// TIA Portal V18 export
// export: Created 2026-06-20T13:30:08.8484285Z, ExportSetting WithDefaults, DisplayName Totally Integrated Automation Portal, DisplayVersion V18, DisplayName TIA Portal Openness, DisplayVersion V18, DisplayName TIA Portal Version Control Interface, DisplayVersion V18, DisplayName STEP 7 Professional, DisplayVersion V18, DisplayName STEP 7 Safety, DisplayVersion V18, DisplayName WinCC Professional, DisplayVersion V18
FUNCTION "FC_HMI_Mirror_PLC1" : Void   // FC40, LAD
{ S7_Optimized_Access := 'TRUE' }
VERSION : 0.1
// stored: AutoNumber true, IsIECCheckEnabled false, SetENOAutomatically false, UDAEnableTagReadback false
BEGIN

REGION Network 1: Mirror V3230_Nuoc_Bon1
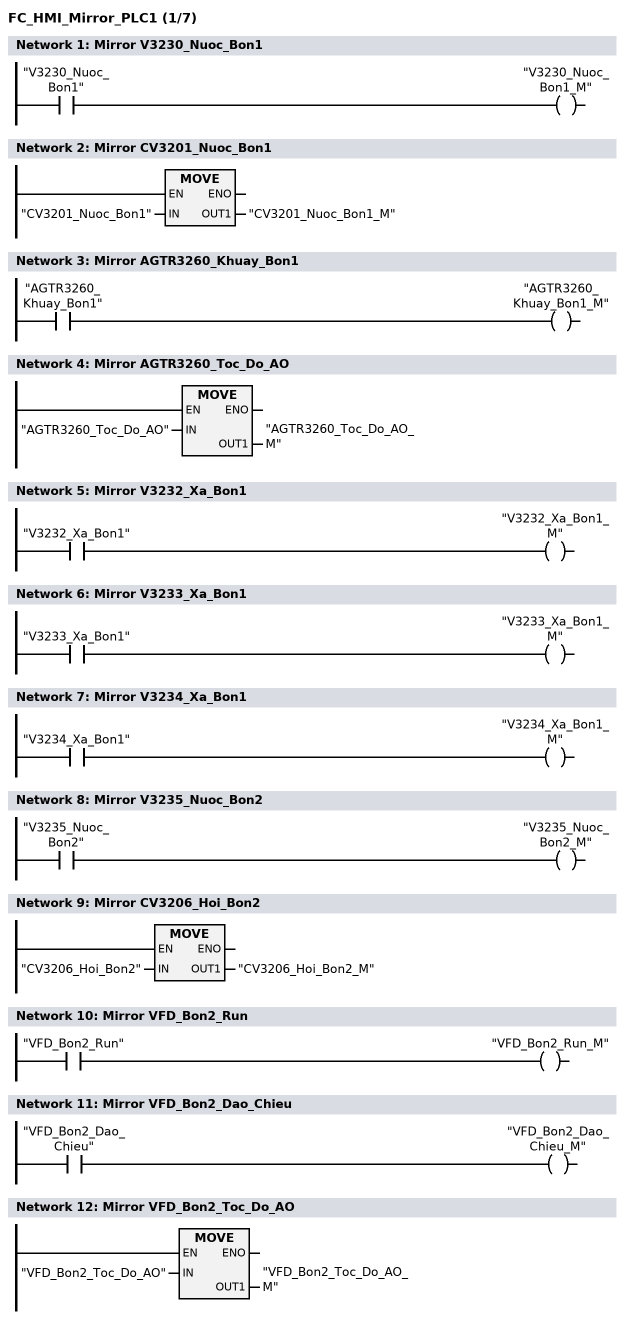
   RUNG wire#powerrail
      Contact( "V3230_Nuoc_Bon1" )
      Coil( "V3230_Nuoc_Bon1_M" )
   END_RUNG
   // the same network as SCL:
   "V3230_Nuoc_Bon1_M" := "V3230_Nuoc_Bon1";
END_REGION

REGION Network 2: Mirror CV3201_Nuoc_Bon1
   RUNG wire#powerrail
      { S7_GenerateENO := "TRUE" } Move(in := "CV3201_Nuoc_Bon1", out1 => "CV3201_Nuoc_Bon1_M")
   END_RUNG
   // the same network as SCL:
   "CV3201_Nuoc_Bon1_M" := "CV3201_Nuoc_Bon1";
END_REGION

REGION Network 3: Mirror AGTR3260_Khuay_Bon1
   RUNG wire#powerrail
      Contact( "AGTR3260_Khuay_Bon1" )
      Coil( "AGTR3260_Khuay_Bon1_M" )
   END_RUNG
   // the same network as SCL:
   "AGTR3260_Khuay_Bon1_M" := "AGTR3260_Khuay_Bon1";
END_REGION

REGION Network 4: Mirror AGTR3260_Toc_Do_AO
   RUNG wire#powerrail
      { S7_GenerateENO := "TRUE" } Move(in := "AGTR3260_Toc_Do_AO", out1 => "AGTR3260_Toc_Do_AO_M")
   END_RUNG
   // the same network as SCL:
   "AGTR3260_Toc_Do_AO_M" := "AGTR3260_Toc_Do_AO";
END_REGION

REGION Network 5: Mirror V3232_Xa_Bon1
   RUNG wire#powerrail
      Contact( "V3232_Xa_Bon1" )
      Coil( "V3232_Xa_Bon1_M" )
   END_RUNG
   // the same network as SCL:
   "V3232_Xa_Bon1_M" := "V3232_Xa_Bon1";
END_REGION

REGION Network 6: Mirror V3233_Xa_Bon1
   RUNG wire#powerrail
      Contact( "V3233_Xa_Bon1" )
      Coil( "V3233_Xa_Bon1_M" )
   END_RUNG
   // the same network as SCL:
   "V3233_Xa_Bon1_M" := "V3233_Xa_Bon1";
END_REGION

REGION Network 7: Mirror V3234_Xa_Bon1
   RUNG wire#powerrail
      Contact( "V3234_Xa_Bon1" )
      Coil( "V3234_Xa_Bon1_M" )
   END_RUNG
   // the same network as SCL:
   "V3234_Xa_Bon1_M" := "V3234_Xa_Bon1";
END_REGION

REGION Network 8: Mirror V3235_Nuoc_Bon2
   RUNG wire#powerrail
      Contact( "V3235_Nuoc_Bon2" )
      Coil( "V3235_Nuoc_Bon2_M" )
   END_RUNG
   // the same network as SCL:
   "V3235_Nuoc_Bon2_M" := "V3235_Nuoc_Bon2";
END_REGION

REGION Network 9: Mirror CV3206_Hoi_Bon2
   RUNG wire#powerrail
      { S7_GenerateENO := "TRUE" } Move(in := "CV3206_Hoi_Bon2", out1 => "CV3206_Hoi_Bon2_M")
   END_RUNG
   // the same network as SCL:
   "CV3206_Hoi_Bon2_M" := "CV3206_Hoi_Bon2";
END_REGION

REGION Network 10: Mirror VFD_Bon2_Run
   RUNG wire#powerrail
      Contact( "VFD_Bon2_Run" )
      Coil( "VFD_Bon2_Run_M" )
   END_RUNG
   // the same network as SCL:
   "VFD_Bon2_Run_M" := "VFD_Bon2_Run";
END_REGION

REGION Network 11: Mirror VFD_Bon2_Dao_Chieu
   RUNG wire#powerrail
      Contact( "VFD_Bon2_Dao_Chieu" )
      Coil( "VFD_Bon2_Dao_Chieu_M" )
   END_RUNG
   // the same network as SCL:
   "VFD_Bon2_Dao_Chieu_M" := "VFD_Bon2_Dao_Chieu";
END_REGION

REGION Network 12: Mirror VFD_Bon2_Toc_Do_AO
   RUNG wire#powerrail
      { S7_GenerateENO := "TRUE" } Move(in := "VFD_Bon2_Toc_Do_AO", out1 => "VFD_Bon2_Toc_Do_AO_M")
   END_RUNG
   // the same network as SCL:
   "VFD_Bon2_Toc_Do_AO_M" := "VFD_Bon2_Toc_Do_AO";
END_REGION

REGION Network 13: Mirror V3237_Xa_Bon2
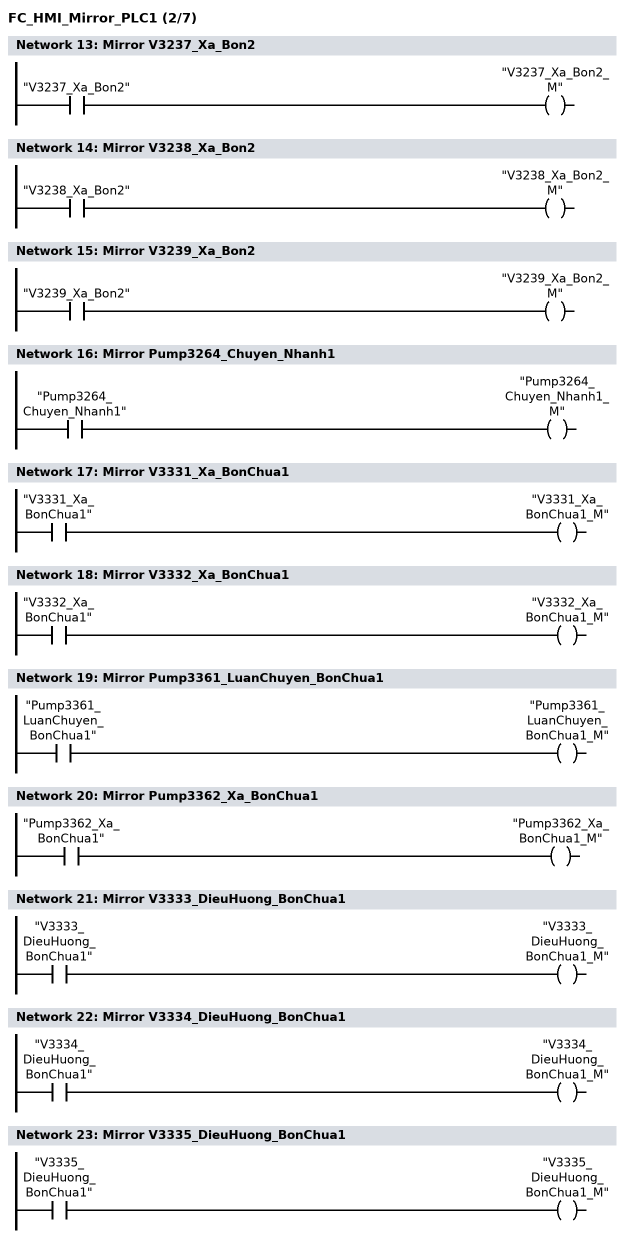
   RUNG wire#powerrail
      Contact( "V3237_Xa_Bon2" )
      Coil( "V3237_Xa_Bon2_M" )
   END_RUNG
   // the same network as SCL:
   "V3237_Xa_Bon2_M" := "V3237_Xa_Bon2";
END_REGION

REGION Network 14: Mirror V3238_Xa_Bon2
   RUNG wire#powerrail
      Contact( "V3238_Xa_Bon2" )
      Coil( "V3238_Xa_Bon2_M" )
   END_RUNG
   // the same network as SCL:
   "V3238_Xa_Bon2_M" := "V3238_Xa_Bon2";
END_REGION

REGION Network 15: Mirror V3239_Xa_Bon2
   RUNG wire#powerrail
      Contact( "V3239_Xa_Bon2" )
      Coil( "V3239_Xa_Bon2_M" )
   END_RUNG
   // the same network as SCL:
   "V3239_Xa_Bon2_M" := "V3239_Xa_Bon2";
END_REGION

REGION Network 16: Mirror Pump3264_Chuyen_Nhanh1
   RUNG wire#powerrail
      Contact( "Pump3264_Chuyen_Nhanh1" )
      Coil( "Pump3264_Chuyen_Nhanh1_M" )
   END_RUNG
   // the same network as SCL:
   "Pump3264_Chuyen_Nhanh1_M" := "Pump3264_Chuyen_Nhanh1";
END_REGION

REGION Network 17: Mirror V3331_Xa_BonChua1
   RUNG wire#powerrail
      Contact( "V3331_Xa_BonChua1" )
      Coil( "V3331_Xa_BonChua1_M" )
   END_RUNG
   // the same network as SCL:
   "V3331_Xa_BonChua1_M" := "V3331_Xa_BonChua1";
END_REGION

REGION Network 18: Mirror V3332_Xa_BonChua1
   RUNG wire#powerrail
      Contact( "V3332_Xa_BonChua1" )
      Coil( "V3332_Xa_BonChua1_M" )
   END_RUNG
   // the same network as SCL:
   "V3332_Xa_BonChua1_M" := "V3332_Xa_BonChua1";
END_REGION

REGION Network 19: Mirror Pump3361_LuanChuyen_BonChua1
   RUNG wire#powerrail
      Contact( "Pump3361_LuanChuyen_BonChua1" )
      Coil( "Pump3361_LuanChuyen_BonChua1_M" )
   END_RUNG
   // the same network as SCL:
   "Pump3361_LuanChuyen_BonChua1_M" := "Pump3361_LuanChuyen_BonChua1";
END_REGION

REGION Network 20: Mirror Pump3362_Xa_BonChua1
   RUNG wire#powerrail
      Contact( "Pump3362_Xa_BonChua1" )
      Coil( "Pump3362_Xa_BonChua1_M" )
   END_RUNG
   // the same network as SCL:
   "Pump3362_Xa_BonChua1_M" := "Pump3362_Xa_BonChua1";
END_REGION

REGION Network 21: Mirror V3333_DieuHuong_BonChua1
   RUNG wire#powerrail
      Contact( "V3333_DieuHuong_BonChua1" )
      Coil( "V3333_DieuHuong_BonChua1_M" )
   END_RUNG
   // the same network as SCL:
   "V3333_DieuHuong_BonChua1_M" := "V3333_DieuHuong_BonChua1";
END_REGION

REGION Network 22: Mirror V3334_DieuHuong_BonChua1
   RUNG wire#powerrail
      Contact( "V3334_DieuHuong_BonChua1" )
      Coil( "V3334_DieuHuong_BonChua1_M" )
   END_RUNG
   // the same network as SCL:
   "V3334_DieuHuong_BonChua1_M" := "V3334_DieuHuong_BonChua1";
END_REGION

REGION Network 23: Mirror V3335_DieuHuong_BonChua1
   RUNG wire#powerrail
      Contact( "V3335_DieuHuong_BonChua1" )
      Coil( "V3335_DieuHuong_BonChua1_M" )
   END_RUNG
   // the same network as SCL:
   "V3335_DieuHuong_BonChua1_M" := "V3335_DieuHuong_BonChua1";
END_REGION

REGION Network 24: Mirror CV3304_Nuoc_Lam_Mat
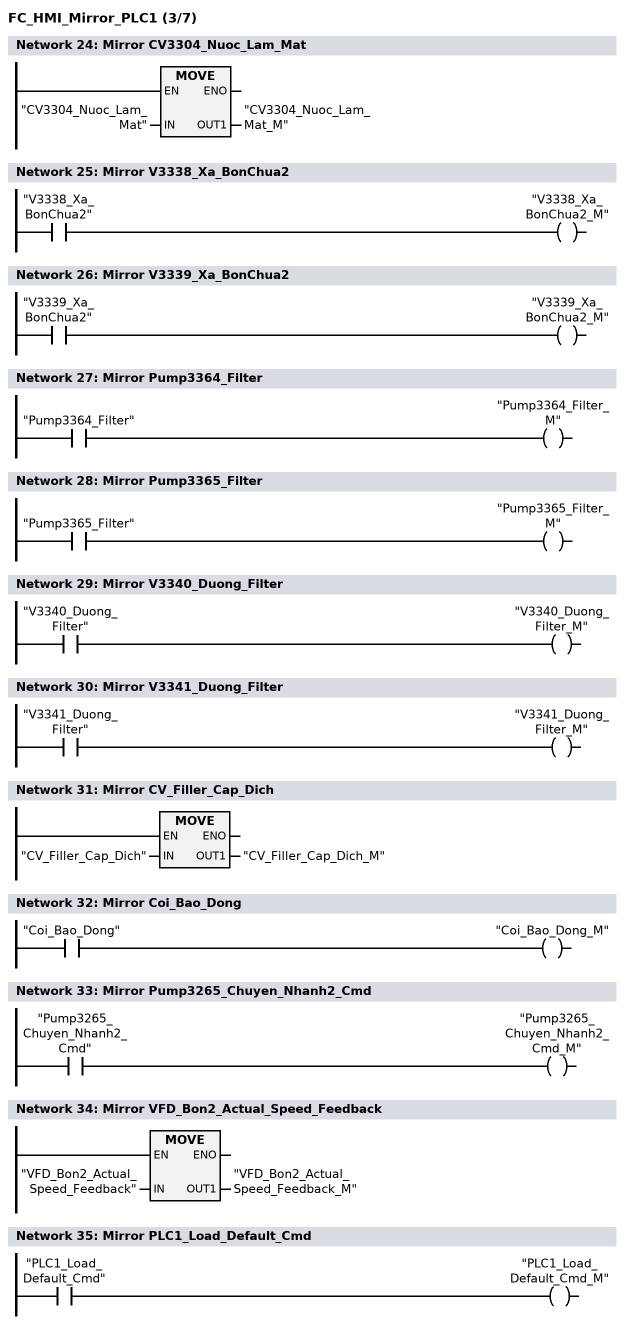
   RUNG wire#powerrail
      { S7_GenerateENO := "TRUE" } Move(in := "CV3304_Nuoc_Lam_Mat", out1 => "CV3304_Nuoc_Lam_Mat_M")
   END_RUNG
   // the same network as SCL:
   "CV3304_Nuoc_Lam_Mat_M" := "CV3304_Nuoc_Lam_Mat";
END_REGION

REGION Network 25: Mirror V3338_Xa_BonChua2
   RUNG wire#powerrail
      Contact( "V3338_Xa_BonChua2" )
      Coil( "V3338_Xa_BonChua2_M" )
   END_RUNG
   // the same network as SCL:
   "V3338_Xa_BonChua2_M" := "V3338_Xa_BonChua2";
END_REGION

REGION Network 26: Mirror V3339_Xa_BonChua2
   RUNG wire#powerrail
      Contact( "V3339_Xa_BonChua2" )
      Coil( "V3339_Xa_BonChua2_M" )
   END_RUNG
   // the same network as SCL:
   "V3339_Xa_BonChua2_M" := "V3339_Xa_BonChua2";
END_REGION

REGION Network 27: Mirror Pump3364_Filter
   RUNG wire#powerrail
      Contact( "Pump3364_Filter" )
      Coil( "Pump3364_Filter_M" )
   END_RUNG
   // the same network as SCL:
   "Pump3364_Filter_M" := "Pump3364_Filter";
END_REGION

REGION Network 28: Mirror Pump3365_Filter
   RUNG wire#powerrail
      Contact( "Pump3365_Filter" )
      Coil( "Pump3365_Filter_M" )
   END_RUNG
   // the same network as SCL:
   "Pump3365_Filter_M" := "Pump3365_Filter";
END_REGION

REGION Network 29: Mirror V3340_Duong_Filter
   RUNG wire#powerrail
      Contact( "V3340_Duong_Filter" )
      Coil( "V3340_Duong_Filter_M" )
   END_RUNG
   // the same network as SCL:
   "V3340_Duong_Filter_M" := "V3340_Duong_Filter";
END_REGION

REGION Network 30: Mirror V3341_Duong_Filter
   RUNG wire#powerrail
      Contact( "V3341_Duong_Filter" )
      Coil( "V3341_Duong_Filter_M" )
   END_RUNG
   // the same network as SCL:
   "V3341_Duong_Filter_M" := "V3341_Duong_Filter";
END_REGION

REGION Network 31: Mirror CV_Filler_Cap_Dich
   RUNG wire#powerrail
      { S7_GenerateENO := "TRUE" } Move(in := "CV_Filler_Cap_Dich", out1 => "CV_Filler_Cap_Dich_M")
   END_RUNG
   // the same network as SCL:
   "CV_Filler_Cap_Dich_M" := "CV_Filler_Cap_Dich";
END_REGION

REGION Network 32: Mirror Coi_Bao_Dong
   RUNG wire#powerrail
      Contact( "Coi_Bao_Dong" )
      Coil( "Coi_Bao_Dong_M" )
   END_RUNG
   // the same network as SCL:
   "Coi_Bao_Dong_M" := "Coi_Bao_Dong";
END_REGION

REGION Network 33: Mirror Pump3265_Chuyen_Nhanh2_Cmd
   RUNG wire#powerrail
      Contact( "Pump3265_Chuyen_Nhanh2_Cmd" )
      Coil( "Pump3265_Chuyen_Nhanh2_Cmd_M" )
   END_RUNG
   // the same network as SCL:
   "Pump3265_Chuyen_Nhanh2_Cmd_M" := "Pump3265_Chuyen_Nhanh2_Cmd";
END_REGION

REGION Network 34: Mirror VFD_Bon2_Actual_Speed_Feedback
   RUNG wire#powerrail
      { S7_GenerateENO := "TRUE" } Move(in := "VFD_Bon2_Actual_Speed_Feedback", out1 => "VFD_Bon2_Actual_Speed_Feedback_M")
   END_RUNG
   // the same network as SCL:
   "VFD_Bon2_Actual_Speed_Feedback_M" := "VFD_Bon2_Actual_Speed_Feedback";
END_REGION

REGION Network 35: Mirror PLC1_Load_Default_Cmd
   RUNG wire#powerrail
      Contact( "PLC1_Load_Default_Cmd" )
      Coil( "PLC1_Load_Default_Cmd_M" )
   END_RUNG
   // the same network as SCL:
   "PLC1_Load_Default_Cmd_M" := "PLC1_Load_Default_Cmd";
END_REGION

REGION Network 36: Quyền Operator
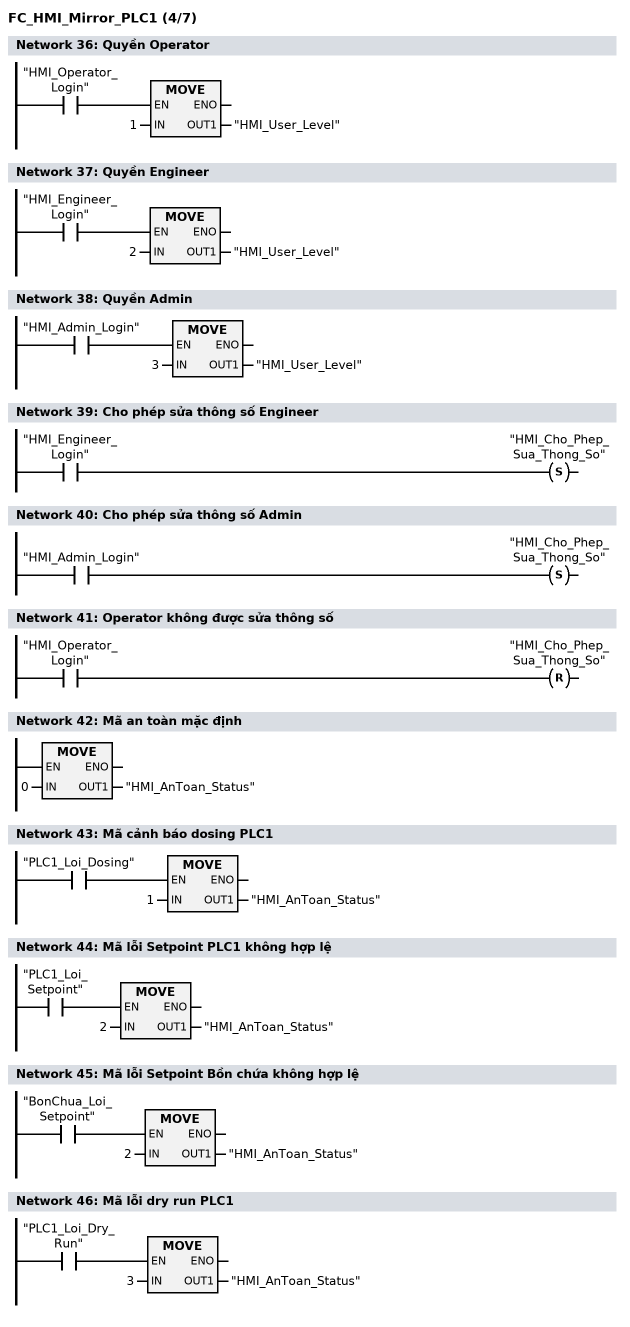
   RUNG wire#powerrail
      Contact( "HMI_Operator_Login" )
      { S7_GenerateENO := "TRUE" } Move(in := 1, out1 => "HMI_User_Level")
   END_RUNG
   // the same network as SCL:
   IF "HMI_Operator_Login" THEN "HMI_User_Level" := 1; END_IF;
END_REGION

REGION Network 37: Quyền Engineer
   RUNG wire#powerrail
      Contact( "HMI_Engineer_Login" )
      { S7_GenerateENO := "TRUE" } Move(in := 2, out1 => "HMI_User_Level")
   END_RUNG
   // the same network as SCL:
   IF "HMI_Engineer_Login" THEN "HMI_User_Level" := 2; END_IF;
END_REGION

REGION Network 38: Quyền Admin
   RUNG wire#powerrail
      Contact( "HMI_Admin_Login" )
      { S7_GenerateENO := "TRUE" } Move(in := 3, out1 => "HMI_User_Level")
   END_RUNG
   // the same network as SCL:
   IF "HMI_Admin_Login" THEN "HMI_User_Level" := 3; END_IF;
END_REGION

REGION Network 39: Cho phép sửa thông số Engineer
   RUNG wire#powerrail
      Contact( "HMI_Engineer_Login" )
      S_Coil( "HMI_Cho_Phep_Sua_Thong_So" )
   END_RUNG
   // the same network as SCL:
   IF "HMI_Engineer_Login" THEN "HMI_Cho_Phep_Sua_Thong_So" := TRUE; END_IF;
END_REGION

REGION Network 40: Cho phép sửa thông số Admin
   RUNG wire#powerrail
      Contact( "HMI_Admin_Login" )
      S_Coil( "HMI_Cho_Phep_Sua_Thong_So" )
   END_RUNG
   // the same network as SCL:
   IF "HMI_Admin_Login" THEN "HMI_Cho_Phep_Sua_Thong_So" := TRUE; END_IF;
END_REGION

REGION Network 41: Operator không được sửa thông số
   RUNG wire#powerrail
      Contact( "HMI_Operator_Login" )
      R_Coil( "HMI_Cho_Phep_Sua_Thong_So" )
   END_RUNG
   // the same network as SCL:
   IF "HMI_Operator_Login" THEN "HMI_Cho_Phep_Sua_Thong_So" := FALSE; END_IF;
END_REGION

REGION Network 42: Mã an toàn mặc định
   RUNG wire#powerrail
      { S7_GenerateENO := "TRUE" } Move(in := 0, out1 => "HMI_AnToan_Status")
   END_RUNG
   // the same network as SCL:
   "HMI_AnToan_Status" := 0;
END_REGION

REGION Network 43: Mã cảnh báo dosing PLC1
   RUNG wire#powerrail
      Contact( "PLC1_Loi_Dosing" )
      { S7_GenerateENO := "TRUE" } Move(in := 1, out1 => "HMI_AnToan_Status")
   END_RUNG
   // the same network as SCL:
   IF "PLC1_Loi_Dosing" THEN "HMI_AnToan_Status" := 1; END_IF;
END_REGION

REGION Network 44: Mã lỗi Setpoint PLC1 không hợp lệ
   RUNG wire#powerrail
      Contact( "PLC1_Loi_Setpoint" )
      { S7_GenerateENO := "TRUE" } Move(in := 2, out1 => "HMI_AnToan_Status")
   END_RUNG
   // the same network as SCL:
   IF "PLC1_Loi_Setpoint" THEN "HMI_AnToan_Status" := 2; END_IF;
END_REGION

REGION Network 45: Mã lỗi Setpoint Bồn chứa không hợp lệ
   RUNG wire#powerrail
      Contact( "BonChua_Loi_Setpoint" )
      { S7_GenerateENO := "TRUE" } Move(in := 2, out1 => "HMI_AnToan_Status")
   END_RUNG
   // the same network as SCL:
   IF "BonChua_Loi_Setpoint" THEN "HMI_AnToan_Status" := 2; END_IF;
END_REGION

REGION Network 46: Mã lỗi dry run PLC1
   RUNG wire#powerrail
      Contact( "PLC1_Loi_Dry_Run" )
      { S7_GenerateENO := "TRUE" } Move(in := 3, out1 => "HMI_AnToan_Status")
   END_RUNG
   // the same network as SCL:
   IF "PLC1_Loi_Dry_Run" THEN "HMI_AnToan_Status" := 3; END_IF;
END_REGION

REGION Network 47: Mã E-Stop ưu tiên cao PLC1
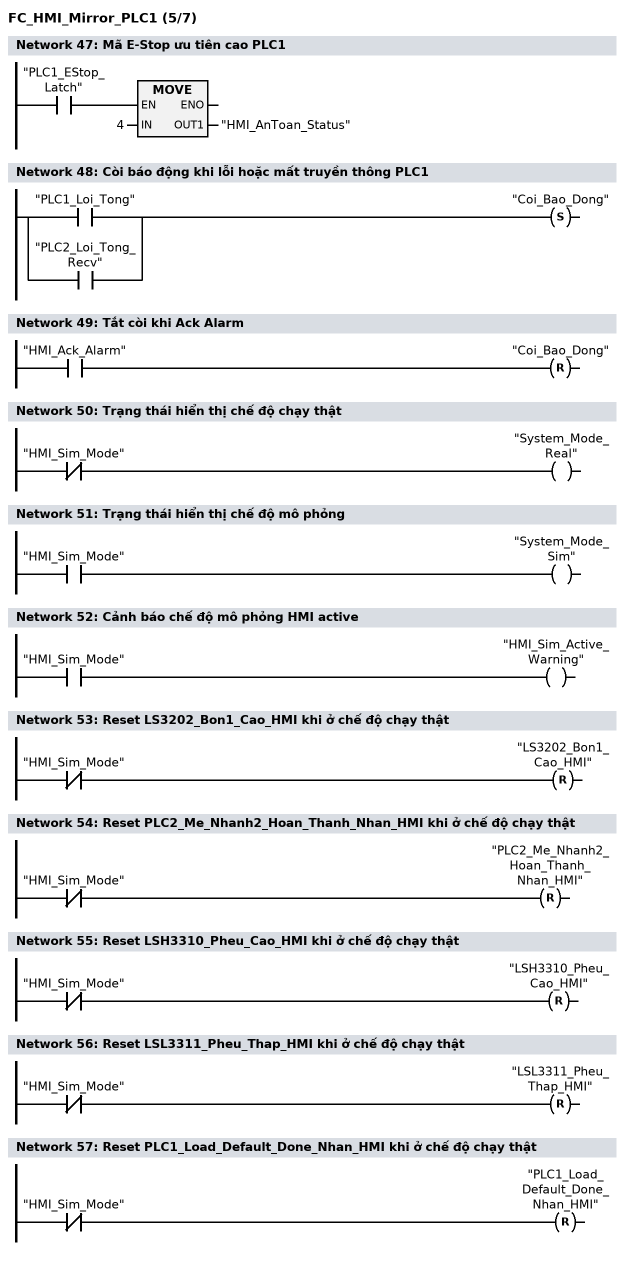
   RUNG wire#powerrail
      Contact( "PLC1_EStop_Latch" )
      { S7_GenerateENO := "TRUE" } Move(in := 4, out1 => "HMI_AnToan_Status")
   END_RUNG
   // the same network as SCL:
   IF "PLC1_EStop_Latch" THEN "HMI_AnToan_Status" := 4; END_IF;
END_REGION

REGION Network 48: Còi báo động khi lỗi hoặc mất truyền thông PLC1
   RUNG wire#powerrail
      Contact( "PLC1_Loi_Tong" )
      wire#w1
      S_Coil( "Coi_Bao_Dong" )
   END_RUNG
   RUNG wire#powerrail
      Contact( "PLC2_Loi_Tong_Recv" )
   END_RUNG wire#w1
   // the same network as SCL:
   IF "PLC1_Loi_Tong" OR "PLC2_Loi_Tong_Recv" THEN "Coi_Bao_Dong" := TRUE; END_IF;
END_REGION

REGION Network 49: Tắt còi khi Ack Alarm
   RUNG wire#powerrail
      Contact( "HMI_Ack_Alarm" )
      R_Coil( "Coi_Bao_Dong" )
   END_RUNG
   // the same network as SCL:
   IF "HMI_Ack_Alarm" THEN "Coi_Bao_Dong" := FALSE; END_IF;
END_REGION

REGION Network 50: Trạng thái hiển thị chế độ chạy thật
   RUNG wire#powerrail
      I_Contact( "HMI_Sim_Mode" )
      Coil( "System_Mode_Real" )
   END_RUNG
   // the same network as SCL:
   "System_Mode_Real" := NOT "HMI_Sim_Mode";
END_REGION

REGION Network 51: Trạng thái hiển thị chế độ mô phỏng
   RUNG wire#powerrail
      Contact( "HMI_Sim_Mode" )
      Coil( "System_Mode_Sim" )
   END_RUNG
   // the same network as SCL:
   "System_Mode_Sim" := "HMI_Sim_Mode";
END_REGION

REGION Network 52: Cảnh báo chế độ mô phỏng HMI active
   RUNG wire#powerrail
      Contact( "HMI_Sim_Mode" )
      Coil( "HMI_Sim_Active_Warning" )
   END_RUNG
   // the same network as SCL:
   "HMI_Sim_Active_Warning" := "HMI_Sim_Mode";
END_REGION

REGION Network 53: Reset LS3202_Bon1_Cao_HMI khi ở chế độ chạy thật
   RUNG wire#powerrail
      I_Contact( "HMI_Sim_Mode" )
      R_Coil( "LS3202_Bon1_Cao_HMI" )
   END_RUNG
   // the same network as SCL:
   IF NOT "HMI_Sim_Mode" THEN "LS3202_Bon1_Cao_HMI" := FALSE; END_IF;
END_REGION

REGION Network 54: Reset PLC2_Me_Nhanh2_Hoan_Thanh_Nhan_HMI khi ở chế độ chạy thật
   RUNG wire#powerrail
      I_Contact( "HMI_Sim_Mode" )
      R_Coil( "PLC2_Me_Nhanh2_Hoan_Thanh_Nhan_HMI" )
   END_RUNG
   // the same network as SCL:
   IF NOT "HMI_Sim_Mode" THEN "PLC2_Me_Nhanh2_Hoan_Thanh_Nhan_HMI" := FALSE; END_IF;
END_REGION

REGION Network 55: Reset LSH3310_Pheu_Cao_HMI khi ở chế độ chạy thật
   RUNG wire#powerrail
      I_Contact( "HMI_Sim_Mode" )
      R_Coil( "LSH3310_Pheu_Cao_HMI" )
   END_RUNG
   // the same network as SCL:
   IF NOT "HMI_Sim_Mode" THEN "LSH3310_Pheu_Cao_HMI" := FALSE; END_IF;
END_REGION

REGION Network 56: Reset LSL3311_Pheu_Thap_HMI khi ở chế độ chạy thật
   RUNG wire#powerrail
      I_Contact( "HMI_Sim_Mode" )
      R_Coil( "LSL3311_Pheu_Thap_HMI" )
   END_RUNG
   // the same network as SCL:
   IF NOT "HMI_Sim_Mode" THEN "LSL3311_Pheu_Thap_HMI" := FALSE; END_IF;
END_REGION

REGION Network 57: Reset PLC1_Load_Default_Done_Nhan_HMI khi ở chế độ chạy thật
   RUNG wire#powerrail
      I_Contact( "HMI_Sim_Mode" )
      R_Coil( "PLC1_Load_Default_Done_Nhan_HMI" )
   END_RUNG
   // the same network as SCL:
   IF NOT "HMI_Sim_Mode" THEN "PLC1_Load_Default_Done_Nhan_HMI" := FALSE; END_IF;
END_REGION

REGION Network 58: Reset FT3200_Bon1_HMI về 0.0 khi ở chế độ chạy thật
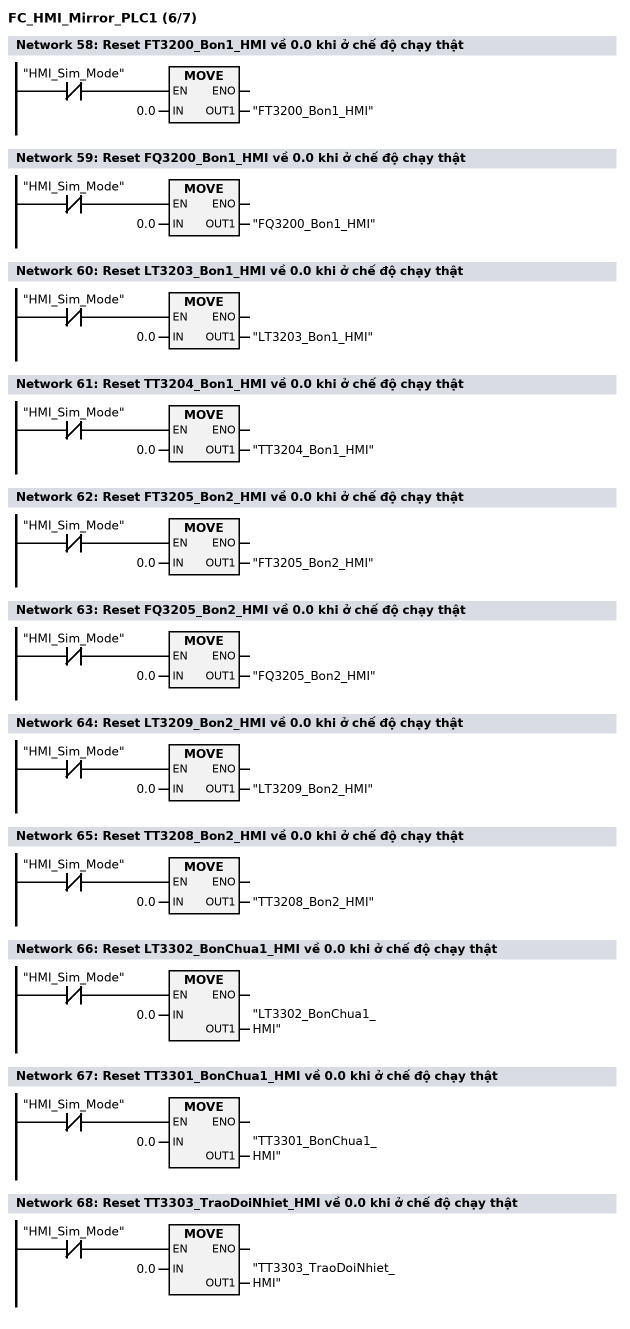
   RUNG wire#powerrail
      I_Contact( "HMI_Sim_Mode" )
      { S7_GenerateENO := "TRUE" } Move(in := 0.0, out1 => "FT3200_Bon1_HMI")
   END_RUNG
   // the same network as SCL:
   IF NOT "HMI_Sim_Mode" THEN "FT3200_Bon1_HMI" := 0.0; END_IF;
END_REGION

REGION Network 59: Reset FQ3200_Bon1_HMI về 0.0 khi ở chế độ chạy thật
   RUNG wire#powerrail
      I_Contact( "HMI_Sim_Mode" )
      { S7_GenerateENO := "TRUE" } Move(in := 0.0, out1 => "FQ3200_Bon1_HMI")
   END_RUNG
   // the same network as SCL:
   IF NOT "HMI_Sim_Mode" THEN "FQ3200_Bon1_HMI" := 0.0; END_IF;
END_REGION

REGION Network 60: Reset LT3203_Bon1_HMI về 0.0 khi ở chế độ chạy thật
   RUNG wire#powerrail
      I_Contact( "HMI_Sim_Mode" )
      { S7_GenerateENO := "TRUE" } Move(in := 0.0, out1 => "LT3203_Bon1_HMI")
   END_RUNG
   // the same network as SCL:
   IF NOT "HMI_Sim_Mode" THEN "LT3203_Bon1_HMI" := 0.0; END_IF;
END_REGION

REGION Network 61: Reset TT3204_Bon1_HMI về 0.0 khi ở chế độ chạy thật
   RUNG wire#powerrail
      I_Contact( "HMI_Sim_Mode" )
      { S7_GenerateENO := "TRUE" } Move(in := 0.0, out1 => "TT3204_Bon1_HMI")
   END_RUNG
   // the same network as SCL:
   IF NOT "HMI_Sim_Mode" THEN "TT3204_Bon1_HMI" := 0.0; END_IF;
END_REGION

REGION Network 62: Reset FT3205_Bon2_HMI về 0.0 khi ở chế độ chạy thật
   RUNG wire#powerrail
      I_Contact( "HMI_Sim_Mode" )
      { S7_GenerateENO := "TRUE" } Move(in := 0.0, out1 => "FT3205_Bon2_HMI")
   END_RUNG
   // the same network as SCL:
   IF NOT "HMI_Sim_Mode" THEN "FT3205_Bon2_HMI" := 0.0; END_IF;
END_REGION

REGION Network 63: Reset FQ3205_Bon2_HMI về 0.0 khi ở chế độ chạy thật
   RUNG wire#powerrail
      I_Contact( "HMI_Sim_Mode" )
      { S7_GenerateENO := "TRUE" } Move(in := 0.0, out1 => "FQ3205_Bon2_HMI")
   END_RUNG
   // the same network as SCL:
   IF NOT "HMI_Sim_Mode" THEN "FQ3205_Bon2_HMI" := 0.0; END_IF;
END_REGION

REGION Network 64: Reset LT3209_Bon2_HMI về 0.0 khi ở chế độ chạy thật
   RUNG wire#powerrail
      I_Contact( "HMI_Sim_Mode" )
      { S7_GenerateENO := "TRUE" } Move(in := 0.0, out1 => "LT3209_Bon2_HMI")
   END_RUNG
   // the same network as SCL:
   IF NOT "HMI_Sim_Mode" THEN "LT3209_Bon2_HMI" := 0.0; END_IF;
END_REGION

REGION Network 65: Reset TT3208_Bon2_HMI về 0.0 khi ở chế độ chạy thật
   RUNG wire#powerrail
      I_Contact( "HMI_Sim_Mode" )
      { S7_GenerateENO := "TRUE" } Move(in := 0.0, out1 => "TT3208_Bon2_HMI")
   END_RUNG
   // the same network as SCL:
   IF NOT "HMI_Sim_Mode" THEN "TT3208_Bon2_HMI" := 0.0; END_IF;
END_REGION

REGION Network 66: Reset LT3302_BonChua1_HMI về 0.0 khi ở chế độ chạy thật
   RUNG wire#powerrail
      I_Contact( "HMI_Sim_Mode" )
      { S7_GenerateENO := "TRUE" } Move(in := 0.0, out1 => "LT3302_BonChua1_HMI")
   END_RUNG
   // the same network as SCL:
   IF NOT "HMI_Sim_Mode" THEN "LT3302_BonChua1_HMI" := 0.0; END_IF;
END_REGION

REGION Network 67: Reset TT3301_BonChua1_HMI về 0.0 khi ở chế độ chạy thật
   RUNG wire#powerrail
      I_Contact( "HMI_Sim_Mode" )
      { S7_GenerateENO := "TRUE" } Move(in := 0.0, out1 => "TT3301_BonChua1_HMI")
   END_RUNG
   // the same network as SCL:
   IF NOT "HMI_Sim_Mode" THEN "TT3301_BonChua1_HMI" := 0.0; END_IF;
END_REGION

REGION Network 68: Reset TT3303_TraoDoiNhiet_HMI về 0.0 khi ở chế độ chạy thật
   RUNG wire#powerrail
      I_Contact( "HMI_Sim_Mode" )
      { S7_GenerateENO := "TRUE" } Move(in := 0.0, out1 => "TT3303_TraoDoiNhiet_HMI")
   END_RUNG
   // the same network as SCL:
   IF NOT "HMI_Sim_Mode" THEN "TT3303_TraoDoiNhiet_HMI" := 0.0; END_IF;
END_REGION

REGION Network 69: Reset LT3307_BonChua2_HMI về 0.0 khi ở chế độ chạy thật
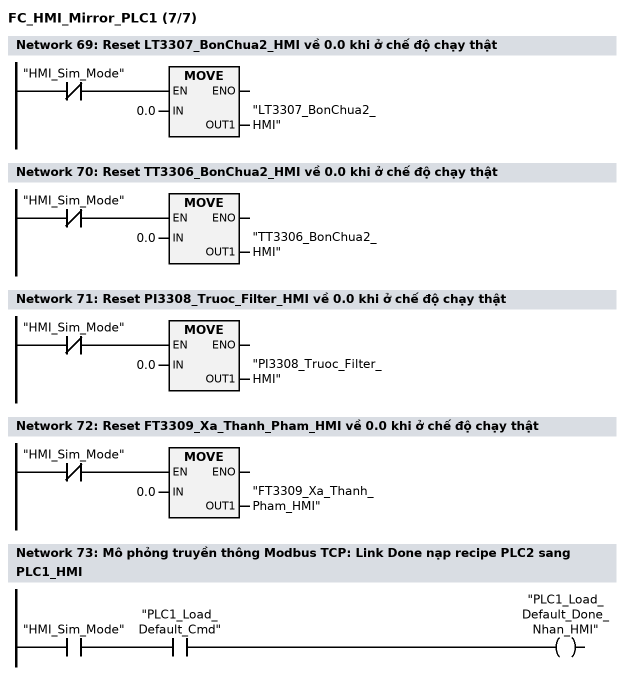
   RUNG wire#powerrail
      I_Contact( "HMI_Sim_Mode" )
      { S7_GenerateENO := "TRUE" } Move(in := 0.0, out1 => "LT3307_BonChua2_HMI")
   END_RUNG
   // the same network as SCL:
   IF NOT "HMI_Sim_Mode" THEN "LT3307_BonChua2_HMI" := 0.0; END_IF;
END_REGION

REGION Network 70: Reset TT3306_BonChua2_HMI về 0.0 khi ở chế độ chạy thật
   RUNG wire#powerrail
      I_Contact( "HMI_Sim_Mode" )
      { S7_GenerateENO := "TRUE" } Move(in := 0.0, out1 => "TT3306_BonChua2_HMI")
   END_RUNG
   // the same network as SCL:
   IF NOT "HMI_Sim_Mode" THEN "TT3306_BonChua2_HMI" := 0.0; END_IF;
END_REGION

REGION Network 71: Reset PI3308_Truoc_Filter_HMI về 0.0 khi ở chế độ chạy thật
   RUNG wire#powerrail
      I_Contact( "HMI_Sim_Mode" )
      { S7_GenerateENO := "TRUE" } Move(in := 0.0, out1 => "PI3308_Truoc_Filter_HMI")
   END_RUNG
   // the same network as SCL:
   IF NOT "HMI_Sim_Mode" THEN "PI3308_Truoc_Filter_HMI" := 0.0; END_IF;
END_REGION

REGION Network 72: Reset FT3309_Xa_Thanh_Pham_HMI về 0.0 khi ở chế độ chạy thật
   RUNG wire#powerrail
      I_Contact( "HMI_Sim_Mode" )
      { S7_GenerateENO := "TRUE" } Move(in := 0.0, out1 => "FT3309_Xa_Thanh_Pham_HMI")
   END_RUNG
   // the same network as SCL:
   IF NOT "HMI_Sim_Mode" THEN "FT3309_Xa_Thanh_Pham_HMI" := 0.0; END_IF;
END_REGION

REGION Network 73: Mô phỏng truyền thông Modbus TCP: Link Done nạp recipe PLC2 sang PLC1_HMI
   RUNG wire#powerrail
      Contact( "HMI_Sim_Mode" )
      Contact( "PLC1_Load_Default_Cmd" )
      Coil( "PLC1_Load_Default_Done_Nhan_HMI" )
   END_RUNG
   // the same network as SCL:
   "PLC1_Load_Default_Done_Nhan_HMI" := "HMI_Sim_Mode" AND "PLC1_Load_Default_Cmd";
END_REGION
END_FUNCTION
